PROGRAM sub_Power
VAR
		fbPowerWerkstatt	:	FB_PowerSocket;
		fbPowerFernseher	:	FB_PowerSocket;
END_VAR

//###################################################################################
//##-----------------------------------POWER---------------------------------------##
//###################################################################################

//--------------------WERKSTATT STECKDOSE----------------------------------
fbPowerWerkstatt.bInputs[0] 	:= gvl_EA.bWID01_2;

fbPowerWerkstatt
(
	bPowerInv_NC	:=	TRUE,
	bInputHA		:=	gvl_HA.bWOD01_2	,
	bOut			=>	gvl_EA.bWOD01_2,
);
//-------------------------------------------------------------------------

//--------------------FERNSEHER STECKDOSE----------------------------------
fbPowerFernseher
(
	bPowerInv_NC	:=	TRUE,
	bInputHA		:=	gvl_HA.bOD02_6,
	bOut			=>	gvl_EA.bOD02_6,
);
//-------------------------------------------------------------------------

END_PROGRAM

(* stored: Version 1.1.0.1, ProductVersion 3.1.4024.4
   POU sub_Power: Id {b9be3092-8a4e-4bbc-8f3f-2431869a4bad}, SpecialFunc None *)
